// TIA Portal V20 export
DATA_BLOCK "DB_Info_From_PCL_Centralizer"   // DB4
{ S7_Optimized_Access := 'TRUE' }
// stored: MemoryReserve 100
   VAR
      Start : Bool;
      Manual_Turn_On_Motor_Caroussel : Bool;
      Manual_Turn_On_Motor_Conveyor_Belt : Bool;
      Water_Foutain_Fail_Functional_Test : Bool;
      Select_Motor_Speed : SInt;
      Carousel_Voltage_Selection : SInt;
   END_VAR
BEGIN
END_DATA_BLOCK
